{attribute addProperty BoxType "EP6224-2022-0016"}
{attribute addProperty Id "DeviceState_Inputs_DeviceAT %I*DeviceState_Inputs_Device_345DC0EE1620DeviceState_InputsAT %I*DeviceState_Inputs_BDC6BEC33240IO_Inputs_ChannelARRAY[0..3] OF EMPTY_STRUCTURE000IO_Outputs_ChannelARRAY[0..3] OF EMPTY_STRUCTURE000WcStateAT %I*WcState_F855686C1620InfoDataAT %I*InfoData_275E3363128160"}
{attribute addProperty CRC "305909798"}
{attribute addProperty SizeInBites "192"}
{attribute addProperty SizeInBytes "24"}
TYPE EP6224_7C2B6CA2 :
STRUCT
	{attribute addProperty Name "DeviceState_Inputs_Device"}
	DeviceState_Inputs_Device : DeviceState_Inputs_Device_345DC0EE;
	{attribute addProperty Name "DeviceState_Inputs"}
	DeviceState_Inputs : DeviceState_Inputs_BDC6BEC3;
	{attribute addProperty Name "IO_Inputs_Channel"}
	IO_Inputs_Channel : ARRAY[0..3] OF EMPTY_STRUCTURE;
	{attribute addProperty Name "IO_Outputs_Channel"}
	IO_Outputs_Channel : ARRAY[0..3] OF EMPTY_STRUCTURE;
	{attribute addProperty Name "WcState"}
	WcState : WcState_F855686C;
	{attribute addProperty Name "InfoData"}
	InfoData : InfoData_275E3363;
END_STRUCT
END_TYPE

(* stored: Version 1.2.0.0, ProductVersion 3.1.4024.9
   DUT EP6224_7C2B6CA2: Id {6da5a986-354d-4103-9ff3-bb5ce593eca2} *)
